{attribute addProperty BoxType "EK1100-0000-0018"}
{attribute addProperty Id "Beckhoff_ELM35xxEK1122Beckhoff_ELM35xxEK1122_B82F516C162A_0001_ELM3502_0000_0016ELM3502_08F8D9E433842.25A_0002_ELM3502_0000_0017ELM3502_08F8D9E433842.25A_0003_ELM3502_0000_0018ELM3502_08F8D9E433842.25A_0004_ELM3502_0000_0019ELM3502_08F8D9E433842.25A_0005_ELM3504_0000_0016ELM3504_B740F21646658.25A_0006_ELM3504_0000_0017ELM3504_B740F21646658.25A_0007_ELM3504_0000_0018ELM3504_B740F21646658.25A_0008_ELM3504_0000_0019ELM3504_B740F21646658.25"}
{attribute addProperty CRC "1173466233"}
{attribute addProperty SizeInBites "3232"}
{attribute addProperty SizeInBytes "404"}
TYPE Beckhoff_ELM35xx_45F1AC79 EXTENDS EK1100_179A0949 :
STRUCT
	{attribute addProperty Name "Beckhoff_ELM35xxEK1122"}
	Beckhoff_ELM35xxEK1122 : Beckhoff_ELM35xxEK1122_B82F516C;
	{attribute addProperty Name "A_0001_ELM3502_0000_0016"}
	A_0001_ELM3502_0000_0016 : ELM3502_08F8D9E4;
	{attribute addProperty Name "A_0002_ELM3502_0000_0017"}
	A_0002_ELM3502_0000_0017 : ELM3502_08F8D9E4;
	{attribute addProperty Name "A_0003_ELM3502_0000_0018"}
	A_0003_ELM3502_0000_0018 : ELM3502_08F8D9E4;
	{attribute addProperty Name "A_0004_ELM3502_0000_0019"}
	A_0004_ELM3502_0000_0019 : ELM3502_08F8D9E4;
	{attribute addProperty Name "A_0005_ELM3504_0000_0016"}
	A_0005_ELM3504_0000_0016 : ELM3504_B740F216;
	{attribute addProperty Name "A_0006_ELM3504_0000_0017"}
	A_0006_ELM3504_0000_0017 : ELM3504_B740F216;
	{attribute addProperty Name "A_0007_ELM3504_0000_0018"}
	A_0007_ELM3504_0000_0018 : ELM3504_B740F216;
	{attribute addProperty Name "A_0008_ELM3504_0000_0019"}
	A_0008_ELM3504_0000_0019 : ELM3504_B740F216;
END_STRUCT
END_TYPE

(* stored: Version 1.2.0.0, ProductVersion 3.1.4024.9
   DUT Beckhoff_ELM35xx_45F1AC79: Id {2c83159d-9499-4814-9754-ed4bf482ce5c} *)
